{attribute 'hide'}
FUNCTION INTERNAL GetFileAgeInSeconds : DINT
VAR_INPUT
  currentUtcTime : Tc2_Utilities.T_FILETIME;
  findFileEntry : Tc2_Utilities.ST_FindFileEntry;
END_VAR
VAR
  _timeLastWriteAccess : Tc2_Utilities.T_ULARGE_INTEGER;
  _fileTimeAsULINT : Tc2_Utilities.T_ULARGE_INTEGER;
  _fileTimeDifference : Tc2_Utilities.T_ULARGE_INTEGER;
END_VAR
VAR CONSTANT
  OneSecondInOneHundredNanoSecondsIntervals : LREAL := 1000*1000*10;
END_VAR

// Local file time
_fileTimeAsULINT.dwLowPart := currentUtcTime.dwLowDateTime;
_fileTimeAsULINT.dwHighPart := currentUtcTime.dwHighDateTime;

// Write access is UTC
_timeLastWriteAccess.dwLowPart := findFileEntry.lastWriteTime.dwLowDateTime;
_timeLastWriteAccess.dwHighPart := findFileEntry.lastWriteTime.dwHighDateTime;
_fileTimeDifference := UInt64Sub64(_fileTimeAsULINT, _timeLastWriteAccess);

GetFileAgeInSeconds := LREAL_TO_DINT(UINT64_TO_LREAL(_fileTimeDifference)/(OneSecondInOneHundredNanoSecondsIntervals));

END_FUNCTION

(* stored: Version 1.1.0.1
   POU GetFileAgeInSeconds: Id {0c3bb6f7-d5ea-49cd-913d-be431f6d46d5}, SpecialFunc None *)
